// TIA Portal V17 export
// export: Created 2023-04-04T13:27:29.5576113Z, ExportSetting WithDefaults, DisplayName Totally Integrated Automation Portal, DisplayVersion V17, DisplayName TIA Portal Openness, DisplayVersion V17, DisplayName TIA Portal Version Control Interface, DisplayVersion V17, DisplayName STEP 7 Professional, DisplayVersion V17, DisplayName STEP 7 Safety, DisplayVersion V17, DisplayName WinCC Advanced, DisplayVersion V17
DATA_BLOCK "RT_INFO_scl_OB30"   // DB325
{ S7_Optimized_Access := 'TRUE' }
VERSION : 0.1
// stored: AutoNumber true, DBAccessibleFromOPCUA true, DBAccessibleFromWebserver true, IsOnlyStoredInLoadMemory false, IsRetainMemResEnabled false, IsWriteProtectedInAS false, MemoryReserve 100
   VAR
      mode { ExternalAccessible := 'False'; ExternalVisible := 'False'; ExternalWritable := 'False'} : UInt := 1;   // Mode 1 = Runtime of a specific OB; 2 = Maximum runtime of a specific OB; 3 = Minimum runtime of a specific OB; 10 = Mean value of the percentage of total runtime used by higher-priority OBs; ...
      obNbr { ExternalAccessible := 'False'; ExternalVisible := 'False'; ExternalWritable := 'False'} : OB_ANY := 1;   // OB to read
      infoData { ExternalAccessible := 'False'; ExternalVisible := 'False'; ExternalWritable := 'False'} : LTime;   // mode 1 --> Runtime in LTIME
      returnValue { ExternalAccessible := 'False'; ExternalVisible := 'False'; ExternalWritable := 'False'} : Int;   // Error information of instruction
   END_VAR
BEGIN
END_DATA_BLOCK
